# EPICS autosave request: 100idPyCRLApp/Db/pyDevCRL_stack_settings.req
file calcout_settings.req P=$(P)$(SYSID):$(OE):stack$(M)_calc
